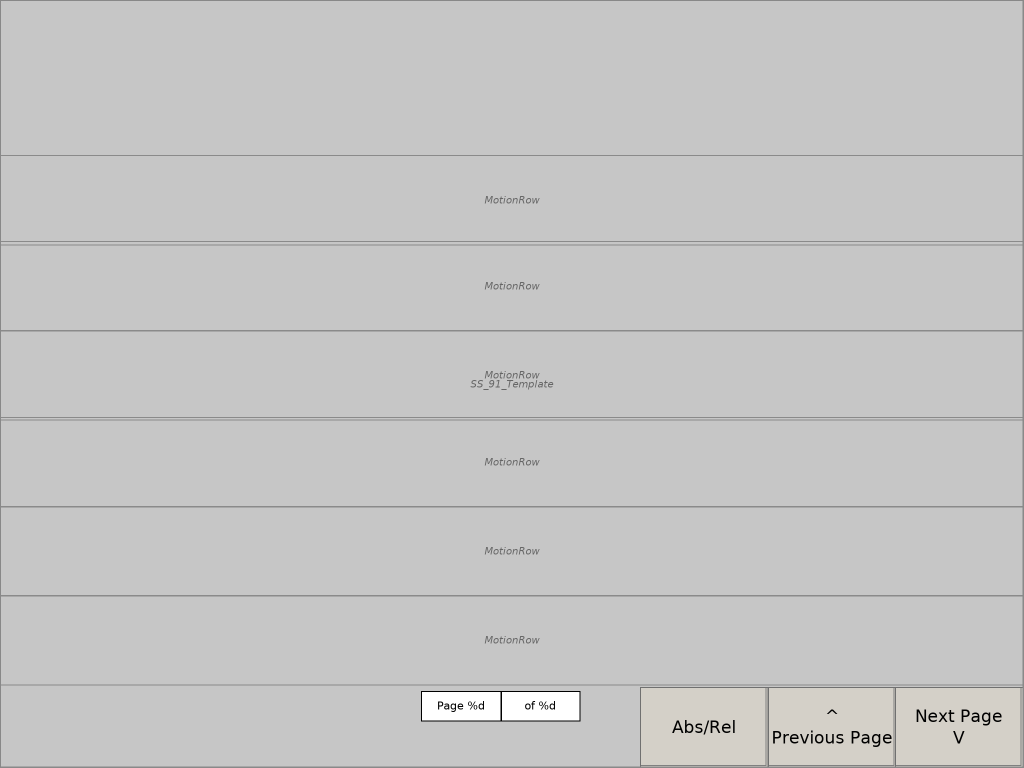
VISUALIZATION SS_99_Motions  // 1024x768
    Frame (0,0 1024x768)
        shows SS_91_Template()
    Frame (0,155 1024x90)
        shows MotionRow(MotionRowInstanceSingle := HMIData.gMotionRows.gMotionRow2, MotionRowButtonsSingle := HMIData.gMotionRowButtons.gMotionRow2btn)
    Frame (0,241 1024x90)
        shows MotionRow(MotionRowInstanceSingle := HMIData.gMotionRows.gMotionRow3, MotionRowButtonsSingle := HMIData.gMotionRowButtons.gMotionRow3btn)
    Frame (0,330 1024x90)
        shows MotionRow(MotionRowInstanceSingle := HMIData.gMotionRows.gMotionRow4, MotionRowButtonsSingle := HMIData.gMotionRowButtons.gMotionRow4btn)
    Frame (0,417 1024x90)
        shows MotionRow(MotionRowInstanceSingle := HMIData.gMotionRows.gMotionRow5, MotionRowButtonsSingle := HMIData.gMotionRowButtons.gMotionRow4btn)
    Frame (0,506 1024x90)
        shows MotionRow(MotionRowInstanceSingle := HMIData.gMotionRows.gMotionRow5, MotionRowButtonsSingle := HMIData.gMotionRowButtons.gMotionRow5btn)
    Frame (0,595 1024x90)
        shows MotionRow(MotionRowInstanceSingle := HMIData.gMotionRows.gMotionRow6, MotionRowButtonsSingle := HMIData.gMotionRowButtons.gMotionRow6btn)
    Button (640,687 128x80), "Abs/Rel", colour toggle: GlobalHMIData.btnAbsMode
        toggle GlobalHMIData.btnAbsMode
    Button (768,687 128x80), "^ Previous Page"
        tap GlobalHMIData.btnPrevPage
    Button (895,687 128x80), "Next Page V"
        tap GlobalHMIData.btnNextPage
    Rectangle (421,691 80x30), "Page %d", text variable: GlobalHMIData.gActivePageNumber
    Rectangle (501,691 79x30), "of %d", text variable: GlobalHMIData.gMaxPageNumber
END_VISUALIZATION

(* stored: Version 1.1.0.1, ProductVersion 3.1.4024.12
   Visu SS_99_Motions: Id {6aba56b7-c6a1-4d88-88c9-c63feb9f8e06} *)
